// TIA Portal V19 export
ORGANIZATION_BLOCK "Main"   // OB1, FBD, ProgramCycle
TITLE = "Main Program Sweep (Cycle)"
{ S7_Optimized_Access := 'TRUE' }
// stored: SetENOAutomatically false
   VAR_INPUT
      Initial_Call : Bool;   // Initial call of this OB
      Remanence : Bool;   // =True, if remanent data are available
   END_VAR
   VAR_TEMP   // added for the SCL form of the ladder/FBD networks
      _w1 : Bool;
   END_VAR
BEGIN

REGION Network 1
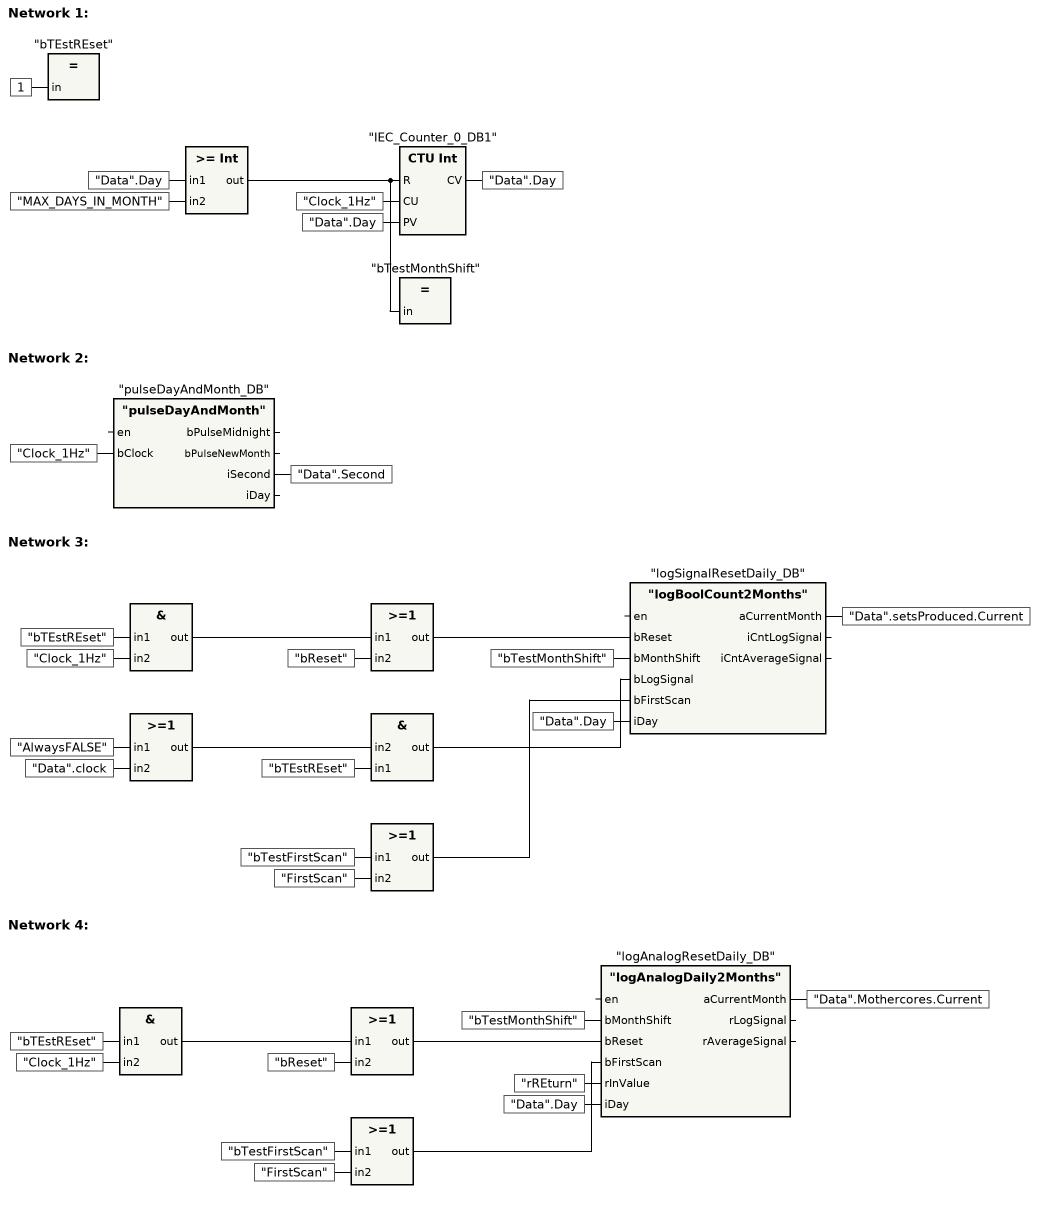
   "bTEstREset" := 1;
   #_w1 := "Data".Day >= "MAX_DAYS_IN_MONTH";
   "IEC_Counter_0_DB1".CTU(R := #_w1, CU := "Clock_1Hz", PV := "Data".Day, CV => "Data".Day);
   "bTestMonthShift" := #_w1;
END_REGION

REGION Network 2
   "pulseDayAndMonth_DB"(bClock := "Clock_1Hz", iSecond => "Data".Second);   // "pulseDayAndMonth"
END_REGION

REGION Network 3
   "logSignalResetDaily_DB"(bReset := ("bTEstREset" AND "Clock_1Hz") OR "bReset",   // "logBoolCount2Months"
                           bMonthShift := "bTestMonthShift",
                           bLogSignal := ("AlwaysFALSE" OR "Data".clock) AND "bTEstREset",
                           bFirstScan := "bTestFirstScan" OR "FirstScan",
                           iDay := "Data".Day,
                           aCurrentMonth => "Data".setsProduced.Current);
END_REGION

REGION Network 4
   "logAnalogResetDaily_DB"(bMonthShift := "bTestMonthShift",   // "logAnalogDaily2Months"
                           bReset := ("bTEstREset" AND "Clock_1Hz") OR "bReset",
                           bFirstScan := "bTestFirstScan" OR "FirstScan",
                           rInValue := "rREturn",
                           iDay := "Data".Day,
                           aCurrentMonth => "Data".Mothercores.Current);
END_REGION

REGION Network 5
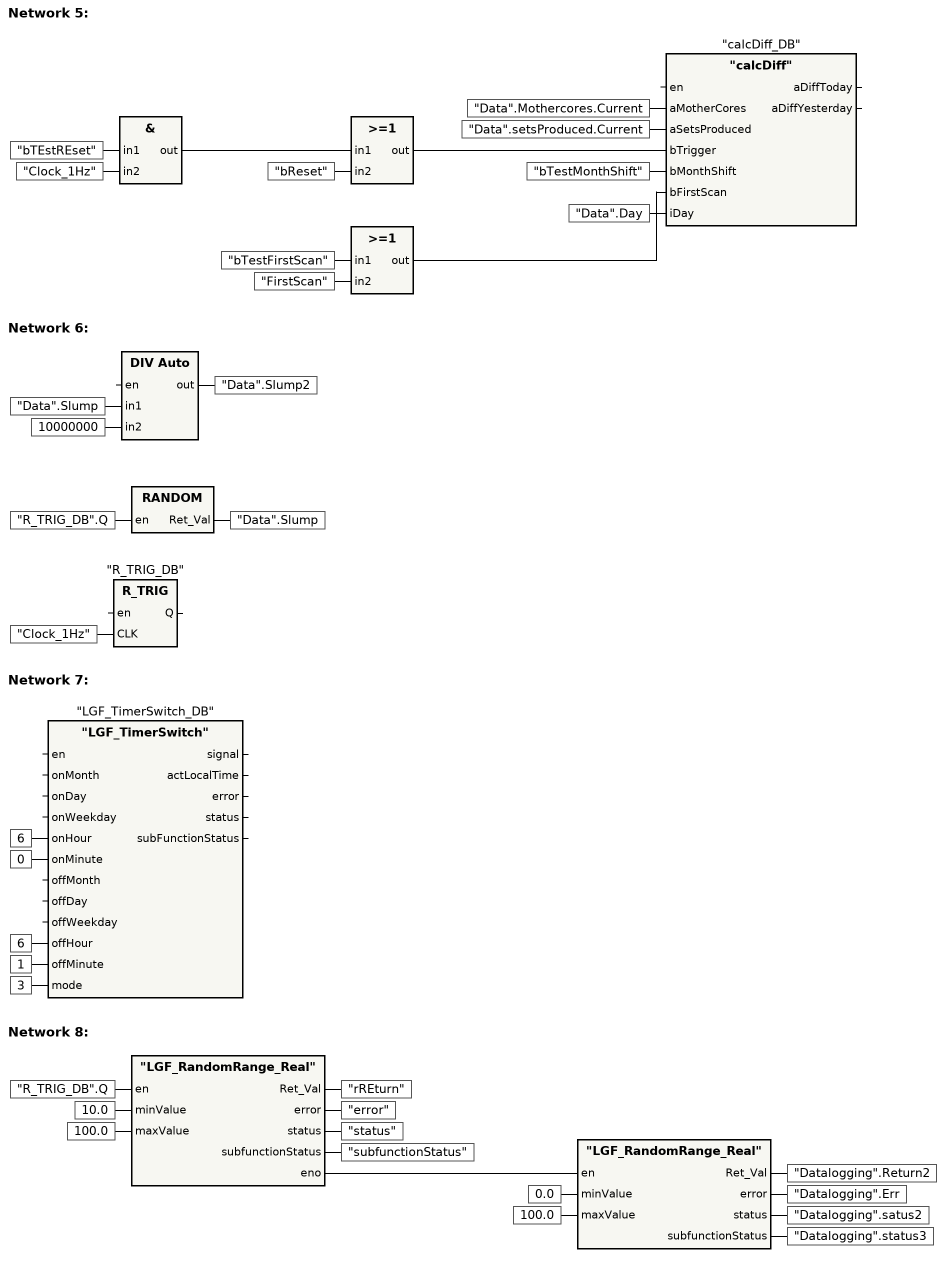
   "calcDiff_DB"(aMotherCores := "Data".Mothercores.Current,   // "calcDiff"
                 aSetsProduced := "Data".setsProduced.Current,
                 bTrigger := ("bTEstREset" AND "Clock_1Hz") OR "bReset",
                 bMonthShift := "bTestMonthShift",
                 bFirstScan := "bTestFirstScan" OR "FirstScan",
                 iDay := "Data".Day);
END_REGION

REGION Network 6
   "Data".Slump2 := "Data".Slump / 10000000;
   IF "R_TRIG_DB".Q THEN "Data".Slump := Random(); END_IF;
   "R_TRIG_DB"(CLK := "Clock_1Hz");   // R_TRIG
END_REGION

REGION Network 7
   "LGF_TimerSwitch_DB"(onHour := 6, onMinute := 0, offHour := 6, offMinute := 1, mode := 3);   // "LGF_TimerSwitch"
END_REGION

REGION Network 8
   "rREturn" := "LGF_RandomRange_Real"(EN := "R_TRIG_DB".Q,
                           minValue := 10.0,
                           maxValue := 100.0,
                           error => "error",
                           status => "status",
                           subfunctionStatus => "subfunctionStatus",
                           ENO => #_w1);
   IF #_w1 THEN
       "Datalogging".Return2 := "LGF_RandomRange_Real"(minValue := 0.0,
                               maxValue := 100.0,
                               error => "Datalogging".Err,
                               status => "Datalogging".satus2,
                               subfunctionStatus => "Datalogging".status3);
   END_IF;
END_REGION

REGION Network 9
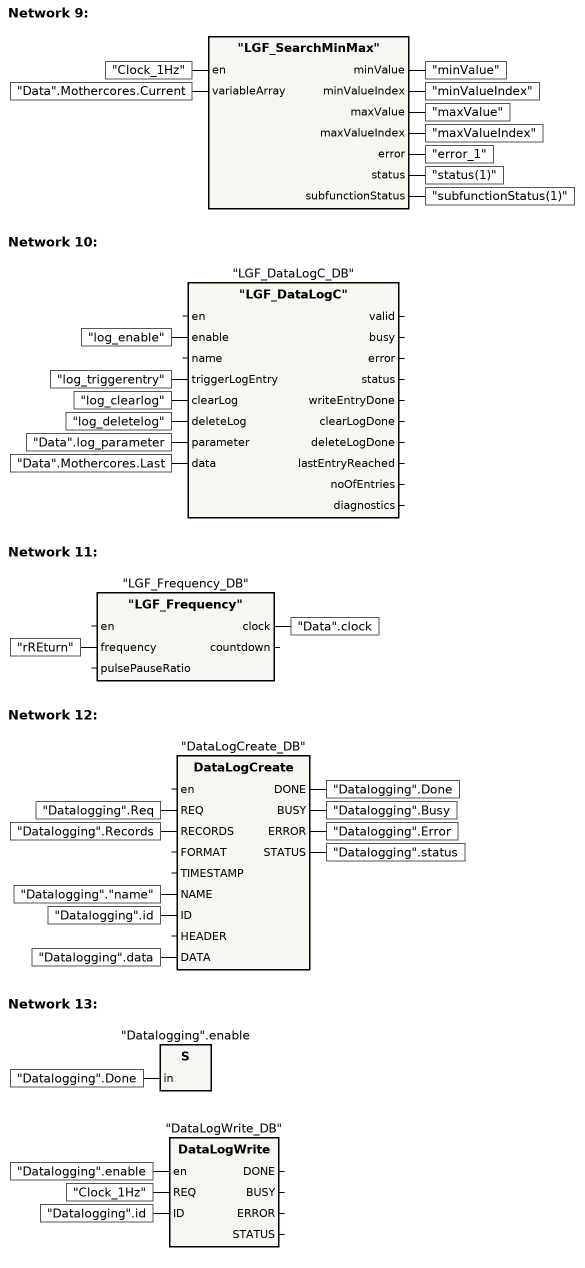
   IF "Clock_1Hz" THEN
       "LGF_SearchMinMax"(variableArray := "Data".Mothercores.Current,
                          minValue => "minValue",
                          minValueIndex => "minValueIndex",
                          maxValue => "maxValue",
                          maxValueIndex => "maxValueIndex",
                          error => "error_1",
                          status => "status(1)",
                          subfunctionStatus => "subfunctionStatus(1)");
   END_IF;
END_REGION

REGION Network 10
   "LGF_DataLogC_DB"(enable := "log_enable",   // "LGF_DataLogC"
                     triggerLogEntry := "log_triggerentry",
                     clearLog := "log_clearlog",
                     deleteLog := "log_deletelog",
                     parameter := "Data".log_parameter,
                     data := "Data".Mothercores.Last);
END_REGION

REGION Network 11
   "LGF_Frequency_DB"(frequency := "rREturn", clock => "Data".clock);   // "LGF_Frequency"
END_REGION

REGION Network 12
   "DataLogCreate_DB"(REQ := "Datalogging".Req,   // DataLogCreate
                      RECORDS := "Datalogging".Records,
                      "NAME" := "Datalogging"."name",
                      ID := "Datalogging".id,
                      DATA := "Datalogging".data,
                      DONE => "Datalogging".Done,
                      BUSY => "Datalogging".Busy,
                      ERROR => "Datalogging".Error,
                      STATUS => "Datalogging".status);
END_REGION

REGION Network 13
   IF "Datalogging".Done THEN "Datalogging".enable := TRUE; END_IF;
   IF "Datalogging".enable THEN
       "DataLogWrite_DB"(REQ := "Clock_1Hz", ID := "Datalogging".id);   // DataLogWrite
   END_IF;
END_REGION

REGION Network 14
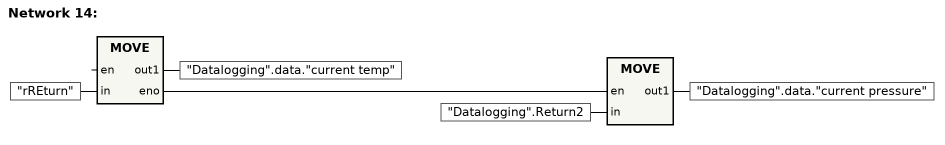
   "Datalogging".data."current temp" := "rREturn";
   "Datalogging".data."current pressure" := "Datalogging".Return2;
END_REGION
END_ORGANIZATION_BLOCK
